FUNCTION_BLOCK Sequenz_1
VAR_INPUT
	Var_1		:BOOL;
	Var_2		:BOOL;
END_VAR
VAR_OUTPUT
	
END_VAR
VAR
	Skill_1			:TestSkill;
END_VAR

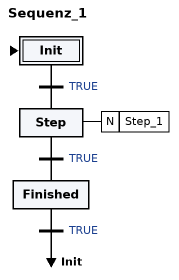
INITIAL_STEP Init:
END_STEP
TRANSITION FROM Init TO Step
    := TRUE;
END_TRANSITION
STEP Step:
    Step_1(N);
END_STEP
TRANSITION FROM Step TO Finished
    := TRUE;
END_TRANSITION
STEP Finished:
END_STEP
TRANSITION FROM Finished TO Init
    := TRUE;
END_TRANSITION

ACTION Step_1:
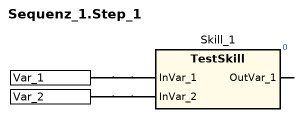
Skill_1(InVar_1 := Var_1, InVar_2 := Var_2); // TestSkill
END_ACTION

END_FUNCTION_BLOCK

(* stored: Version 1.1.0.1
   POU Sequenz_1: Id {6972fbed-b1f6-4cdd-9b33-a67161d238ce}, SpecialFunc None
   Action Step_1: Id {a027a849-00b6-4612-b837-9d30c3f0d9c9} *)
